# EPICS IOC start-up script: test/startup/st.mcu007-PTP-B02.iocsh
epicsEnvSet("MOTOR_PORT",    "$(SM_MOTOR_PORT=MCU1)")
epicsEnvSet("IPADDR",        "$(SM_IPADDR=172.30.38.37)")
epicsEnvSet("IPPORT",        "$(SM_IPPORT=48898)")
epicsEnvSet("AMSNETIDIOC",   "172.30.38.12.1.1")
epicsEnvSet("ASYN_PORT",     "$(SM_ASYN_PORT=MC_CPU1)")
epicsEnvSet("PREFIX",        "$(SM_PREFIX=LabS-MCAG:MC-MCU-07:)")
epicsEnvSet("PREC",          "$(SM_PREC=3)")
epicsEnvSet("SM_NOAXES",     "1")
epicsEnvSet("ECM_OPTIONS",   "adsPort=852;amsNetIdRemote=192.168.88.57.1.1;amsNetIdLocal=$(AMSNETIDIOC)"

# Do not start the poller yet
epicsEnvSet("ECM_MOVINGPOLLPERIOD", "0")
epicsEnvSet("ECM_IDLEPOLLPERIOD",   "0")

< ethercatmcController.iocsh
< ethercatmcEL6688-PTP.iocsh
< ethercatmcEL6688-EL1252-PTP.iocsh

#
# Axis 1
#
epicsEnvSet("AXISCONFIG",    "")
epicsEnvSet("MOTOR_NAME",    "$(SM_MOTOR_NAME=m1)")
epicsEnvSet("AXIS_NO",       "$(SM_AXIS_NO=1)")
epicsEnvSet("DESC",          "$(SM_DESC=DESC)")
epicsEnvSet("EGU",           "$(SM_EGU=EGU)")
epicsEnvSet("RAWENCSTEP_ADEL", 0)
epicsEnvSet("RAWENCSTEP_MDEL", 0)
< ethercatmcIndexerAxis.iocsh
< ethercatmcAxisdebug.iocsh

# Raw steps and velocity
< ethercatmcRawMtrEnc.iocsh

# PLCopen state machine
< ethercatmcPLCopenStateMachine.iocsh

# Predefined Positions
epicsEnvSet("NVL",           "")
epicsEnvSet("EGU",           "")
< ethercatmcDefPos.iocsh
< ethercatmcRawMtrEnc.iocsh

#####################################################
# EL1252, first channel, CHNO == 0
epicsEnvSet("CHNO",     "0")
< ethercatmcEL1252-OneChannel.iocsh
# EL1252, second channel, CHNO == 1
epicsEnvSet("CHNO",     "1")
< ethercatmcEL1252-OneChannel.iocsh

#####################################################
# PTP with ExtSync
< ethercatmcEL6688-PTP.iocsh

# Analog input, copy of TS_NS for testing
epicsEnvSet("CHNO",             "0")
epicsEnvSet("ASYNPARAMNAME",    "TS_NS_AI")
epicsEnvSet("P",                "$(PREFIX)")
epicsEnvSet("R",                "TS_NS_AI")
< ethercatmcAnalogInput.iocsh

#
# Start polling, values are in millisconds
#
epicsEnvSet("MOVINGPOLLPERIOD", "9")
epicsEnvSet("IDLEPOLLPERIOD",   "100")
ethercatmcStartPoller("$(MOTOR_PORT)", "$(MOVINGPOLLPERIOD)", "$(IDLEPOLLPERIOD)")
